(* PLC project Unnamed, Unknown Unnamed 1 *)
(* stored: creationDateTime 2025-11-06T09:56:44, modificationDateTime 2025-11-07T13:27:40 *)

TYPE TrafficLightStruct : STRUCT
  Safe : BOOL := True;
  LightRed : BOOL := False;
  LightGreen : BOOL := False;
  LightYellow : BOOL := False;
END_STRUCT;
END_TYPE

TYPE CrossWalkStruct : STRUCT
  Safe : BOOL := True;
  WalkLight : BOOL := False;
  DontWalkLight : BOOL := False;
END_STRUCT;
END_TYPE

TYPE InputMapStruct : STRUCT
  StartButton : BOOL := False;
  StopButton : BOOL := True;
  ResetButton : BOOL := False;
  CrossButton : BOOL := False;
  RedLightSensor : BOOL := True;
  GreenLightSensor : BOOL := True;
  YellowLightSensor : BOOL := True;
  WalkLightSensor : BOOL := True;
  DontWalkLightSensor : BOOL := True;
END_STRUCT;
END_TYPE

PROGRAM input_mapping0
  VAR_EXTERNAL
    DI_PB1 : BOOL;
    DI_PB2 : BOOL;
    DI_PB3 : BOOL;
    DI_PB4 : BOOL;
    DI_LightSensor1 : BOOL;
    DI_LightSensor2 : BOOL;
    DI_LightSensor3 : BOOL;
    DI_LightSensor4 : BOOL;
    DI_LightSensor5 : BOOL;
    InputMapGlobal : InputMapStruct;
  END_VAR

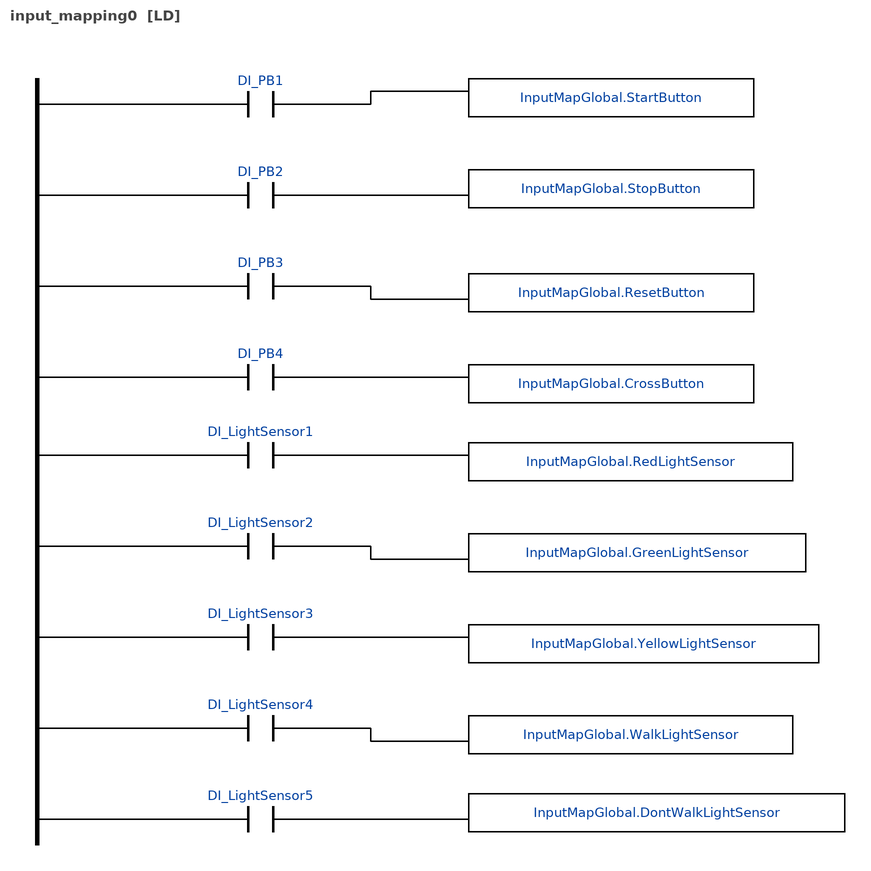
(* LD diagram, written out as Structured Text *)
InputMapGlobal.StartButton := DI_PB1;
InputMapGlobal.StopButton := DI_PB2;
InputMapGlobal.CrossButton := DI_PB4;
InputMapGlobal.RedLightSensor := DI_LightSensor1;
InputMapGlobal.GreenLightSensor := DI_LightSensor2;
InputMapGlobal.ResetButton := DI_PB3;
InputMapGlobal.YellowLightSensor := DI_LightSensor3;
InputMapGlobal.WalkLightSensor := DI_LightSensor4;
InputMapGlobal.DontWalkLightSensor := DI_LightSensor5;
END_PROGRAM

PROGRAM SystemControl
  VAR_EXTERNAL
    InputMapGlobal : InputMapStruct;
    Safe : BOOL;
  END_VAR
  VAR
    StartButton : BOOL;
    StopButton : BOOL;
  END_VAR
  VAR_EXTERNAL
    Running : BOOL;
  END_VAR

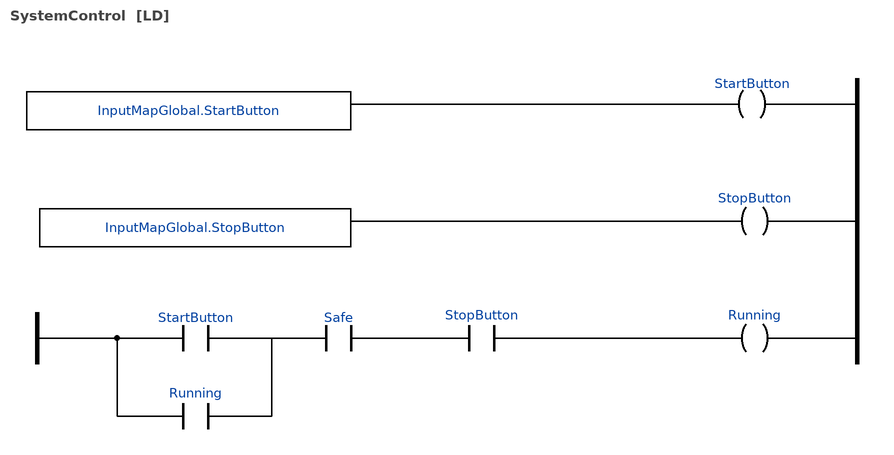
(* LD diagram, written out as Structured Text *)
StartButton := InputMapGlobal.StartButton;
StopButton := InputMapGlobal.StopButton;
Running := (StartButton OR Running) AND Safe AND StopButton;
END_PROGRAM

FUNCTION_BLOCK Flasher
  VAR_INPUT
    OnTime : TIME;
    OffTime : TIME;
  END_VAR
  VAR
    TON0 : TON;
    TOF0 : TOF;
  END_VAR
  VAR_OUTPUT
    F_On : BOOL;
  END_VAR

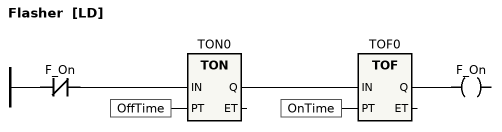
(* LD diagram, written out as Structured Text *)
TON0(IN := NOT F_On, PT := OffTime);
TOF0(IN := TON0.Q, PT := OnTime);
F_On := TOF0.Q;
END_FUNCTION_BLOCK

PROGRAM TrafficLightControl
  VAR_EXTERNAL
    Running : BOOL;
    Safe : BOOL;
    InputMapGlobal : InputMapStruct;
    TrafficLightState : TrafficLightStruct;
  END_VAR
  VAR
    LightCycle : BOOL := False;
    BlinkCycle : BOOL := False;
  END_VAR
  VAR
    Fault_RedLight AT %QX1.0 : BOOL := False;
    Fault_GreenLight AT %QX1.1 : BOOL := False;
    Fault_YellowLight AT %QX1.2 : BOOL := False;
  END_VAR
  VAR
    RedLight : BOOL := False;
    GreenLight : BOOL := False;
    YellowLight : BOOL := False;
    Reset : BOOL := False;
    ResetButton : BOOL := False;
    RedLightSensor : BOOL := False;
    GreenLightSensor : BOOL := False;
    YellowLightSensor : BOOL := False;
    T_YellowLight : TON;
    T_RedLight : TON;
    T_GreenLight : TON;
    Flasher1 : Flasher;
  END_VAR
  VAR  (* added by the conversion: wires and edge detectors of the diagram *)
    R_TRIG1 : R_TRIG;
  END_VAR

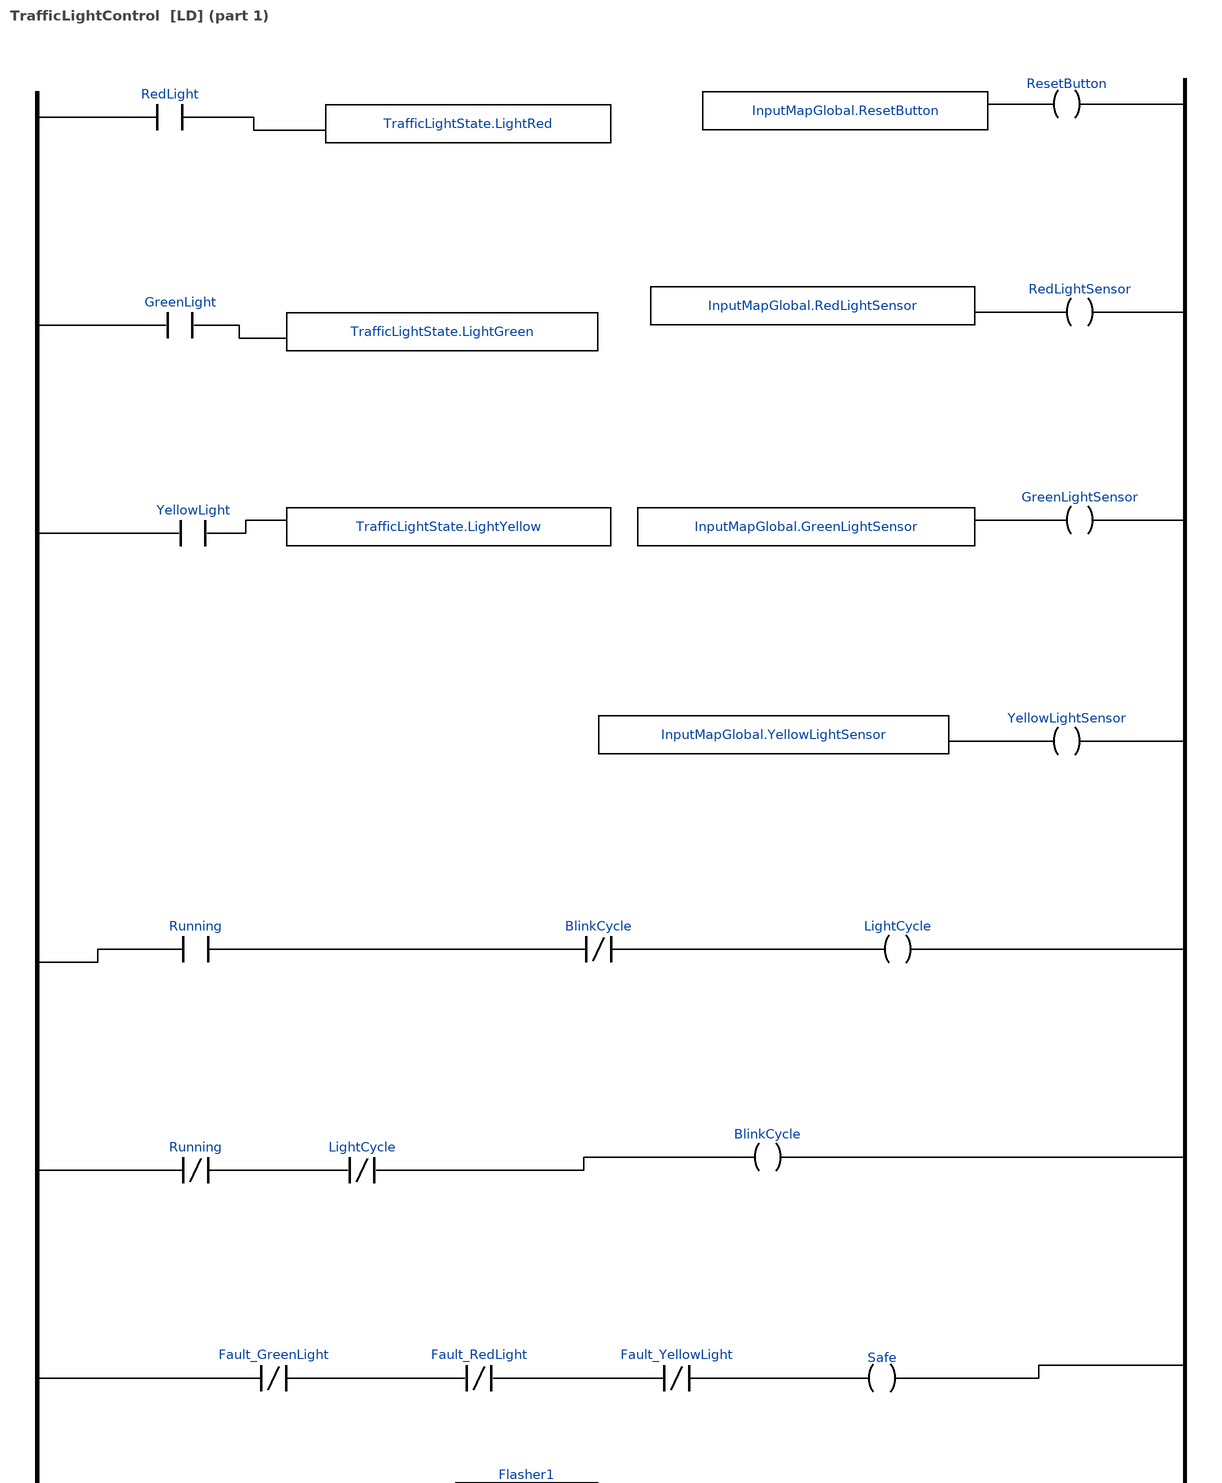
(* LD diagram, written out as Structured Text *)
ResetButton := InputMapGlobal.ResetButton;
RedLightSensor := InputMapGlobal.RedLightSensor;
GreenLightSensor := InputMapGlobal.GreenLightSensor;
YellowLightSensor := InputMapGlobal.YellowLightSensor;
LightCycle := Running AND NOT BlinkCycle;
BlinkCycle := NOT Running AND NOT LightCycle;
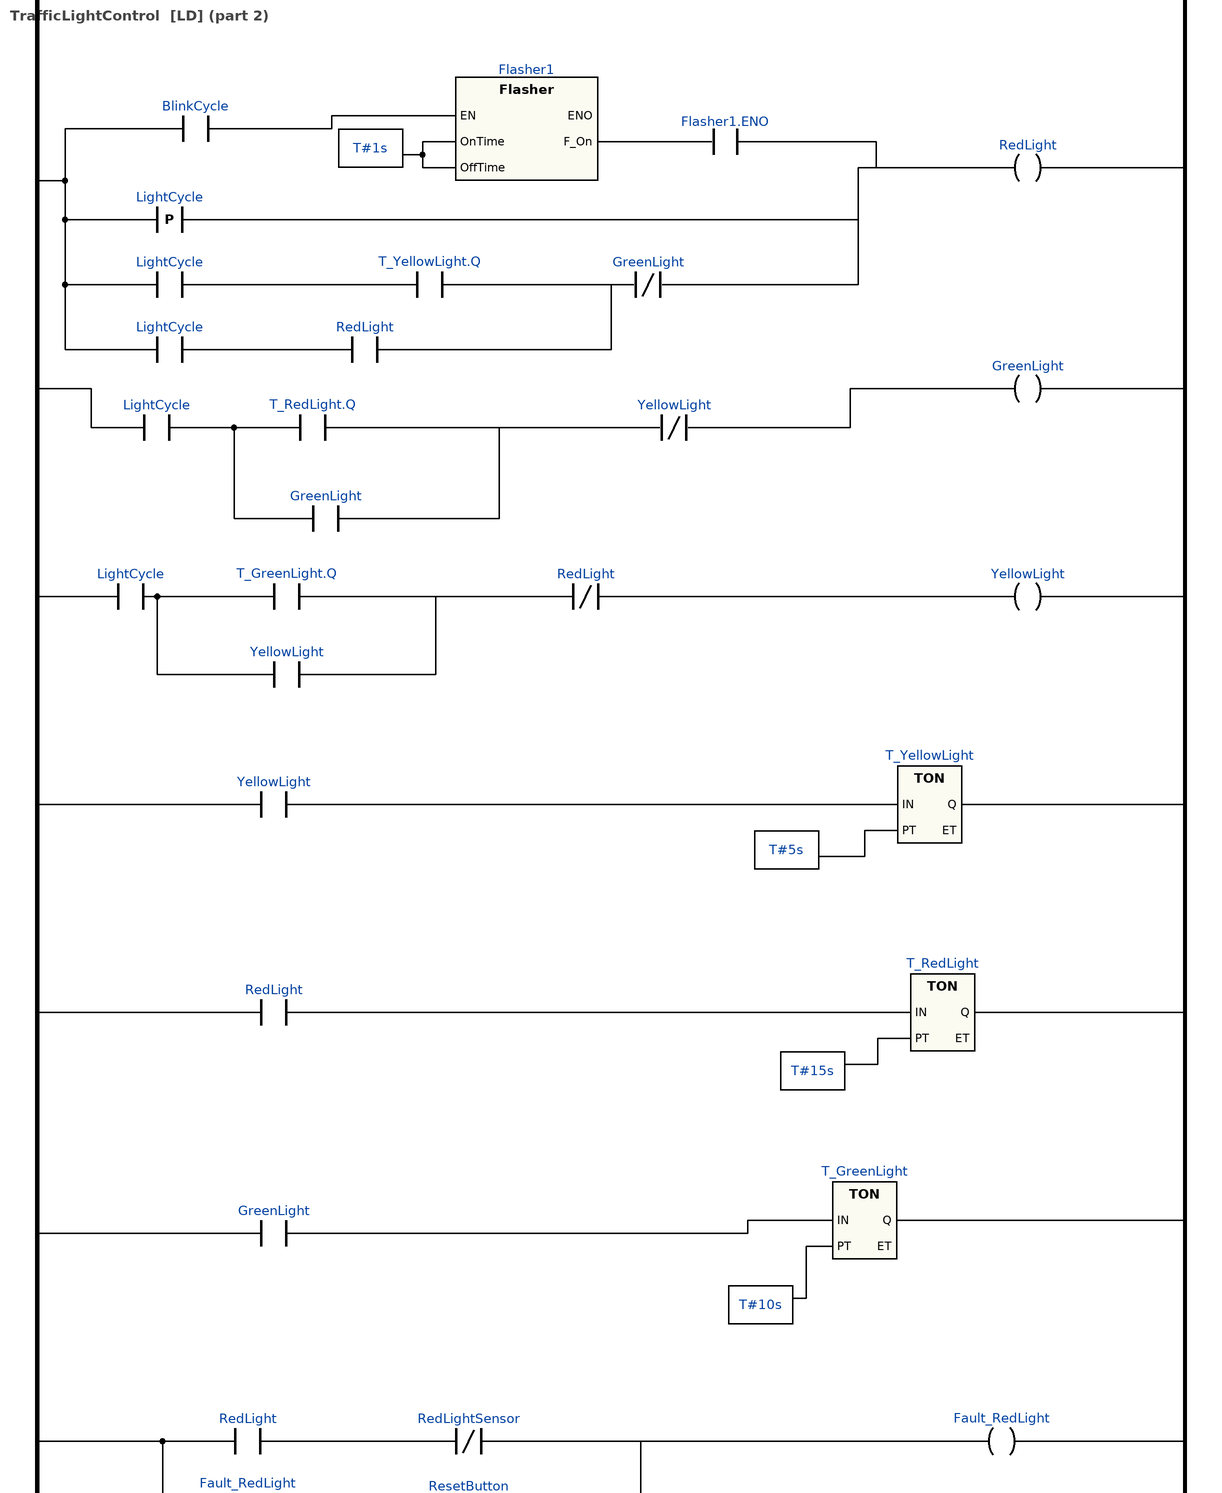
GreenLight := LightCycle AND (T_RedLight.Q OR GreenLight) AND NOT YellowLight;
YellowLight := LightCycle AND (T_GreenLight.Q OR YellowLight) AND NOT RedLight;
R_TRIG1(CLK := LightCycle);
Flasher1(EN := BlinkCycle, OnTime := T#1s, OffTime := T#1s);
RedLight := R_TRIG1.Q OR LightCycle AND (T_YellowLight.Q OR RedLight) AND NOT GreenLight OR Flasher1.F_On AND Flasher1.ENO;
Fault_RedLight := RedLight AND NOT RedLightSensor OR Fault_RedLight AND NOT ResetButton;
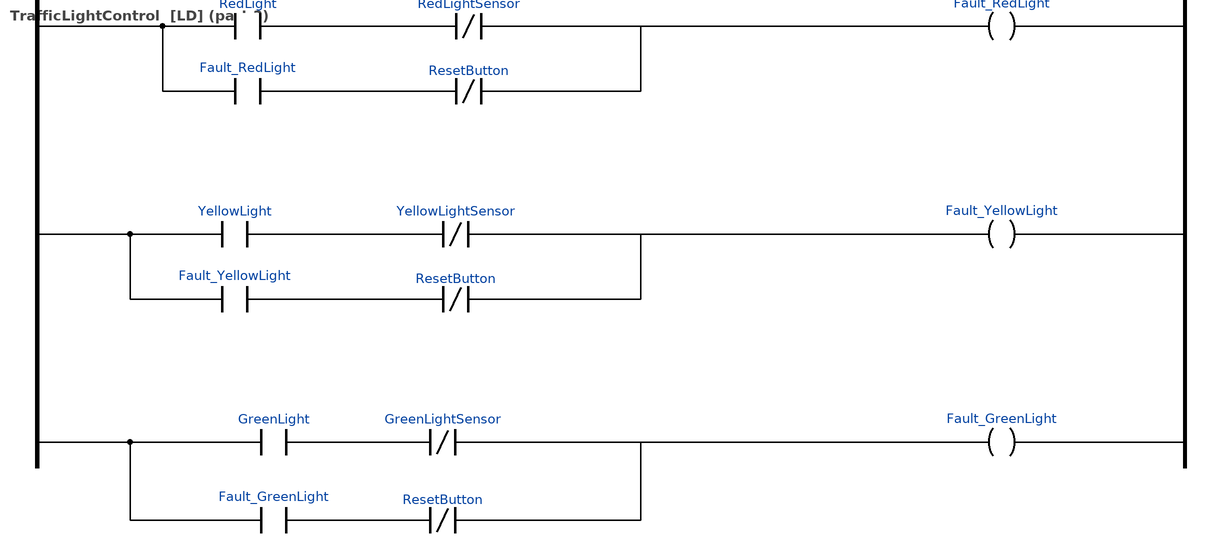
Fault_YellowLight := YellowLight AND NOT YellowLightSensor OR Fault_YellowLight AND NOT ResetButton;
Fault_GreenLight := GreenLight AND NOT GreenLightSensor OR Fault_GreenLight AND NOT ResetButton;
Safe := NOT Fault_GreenLight AND NOT Fault_RedLight AND NOT Fault_YellowLight;
TrafficLightState.LightRed := RedLight;
TrafficLightState.LightGreen := GreenLight;
TrafficLightState.LightYellow := YellowLight;
T_YellowLight(IN := YellowLight, PT := T#5s);
T_RedLight(IN := RedLight, PT := T#15s);
T_GreenLight(IN := GreenLight, PT := T#10s);
END_PROGRAM

PROGRAM CrosswalkControl
  VAR_EXTERNAL
    InputMapGlobal : InputMapStruct;
    CrossWalkState : CrossWalkStruct;
    TrafficLightState : TrafficLightStruct;
    Running : BOOL;
    Safe : BOOL;
  END_VAR
  VAR
    CrosswalkButton : BOOL := False;
    ResetButton : BOOL := False;
    WalkLight : BOOL := False;
    DontWalkLight : BOOL := False;
    CrosswalkSequence : BOOL := False;
    CrosswalkSequence_End : BOOL := False;
    WalkLightFault : BOOL := False;
    DontWalkLightFault : BOOL := False;
    WaitForWalk : BOOL := False;
    Walk : BOOL := False;
    StopWalk : BOOL := False;
    RedLight : BOOL := False;
    GreenLight : BOOL := False;
    T_Walk : TON;
    Flasher0 : Flasher;
    DontWalkLightSensor : BOOL;
    WalkLightSensor : BOOL;
  END_VAR
  VAR  (* added by the conversion: wires and edge detectors of the diagram *)
    R_TRIG1 : R_TRIG;
    R_TRIG2 : R_TRIG;
    R_TRIG3 : R_TRIG;
  END_VAR

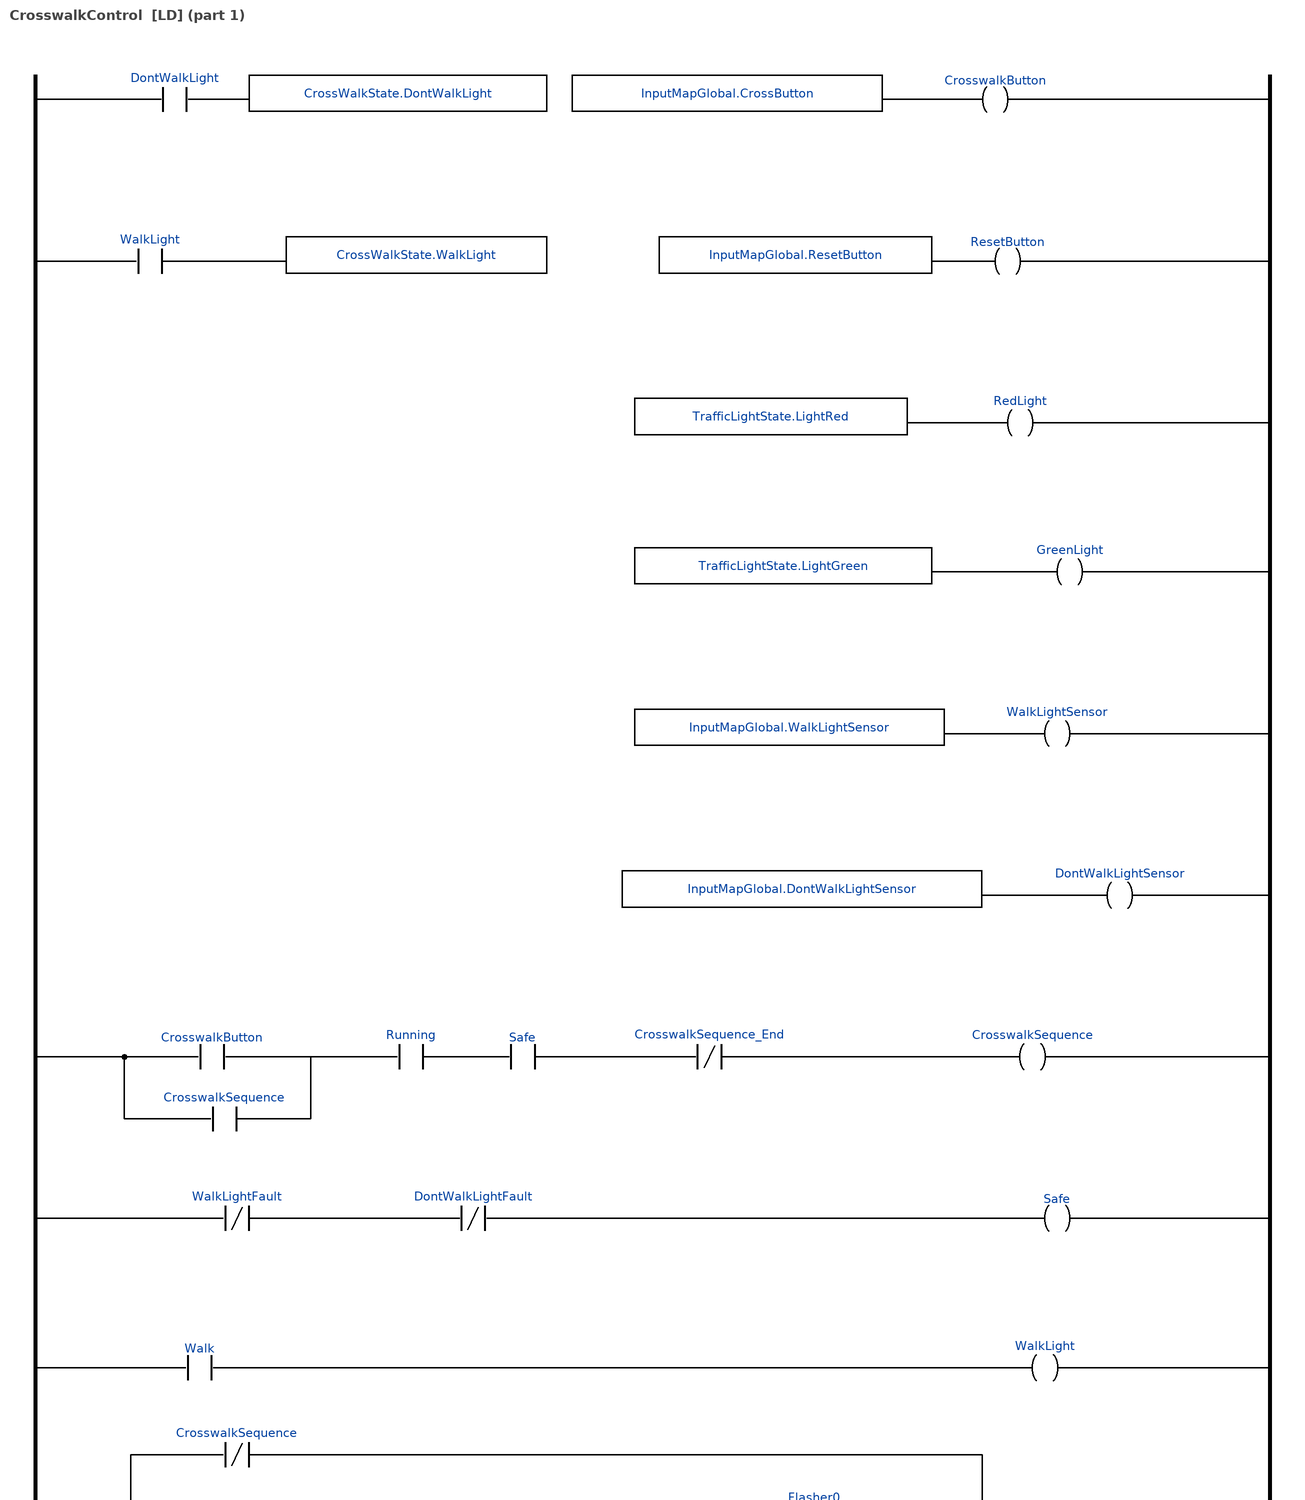
(* LD diagram, written out as Structured Text *)
CrosswalkButton := InputMapGlobal.CrossButton;
ResetButton := InputMapGlobal.ResetButton;
CrossWalkState.DontWalkLight := DontWalkLight;
CrossWalkState.WalkLight := WalkLight;
CrosswalkSequence := (CrosswalkButton OR CrosswalkSequence) AND Running AND Safe AND NOT CrosswalkSequence_End;
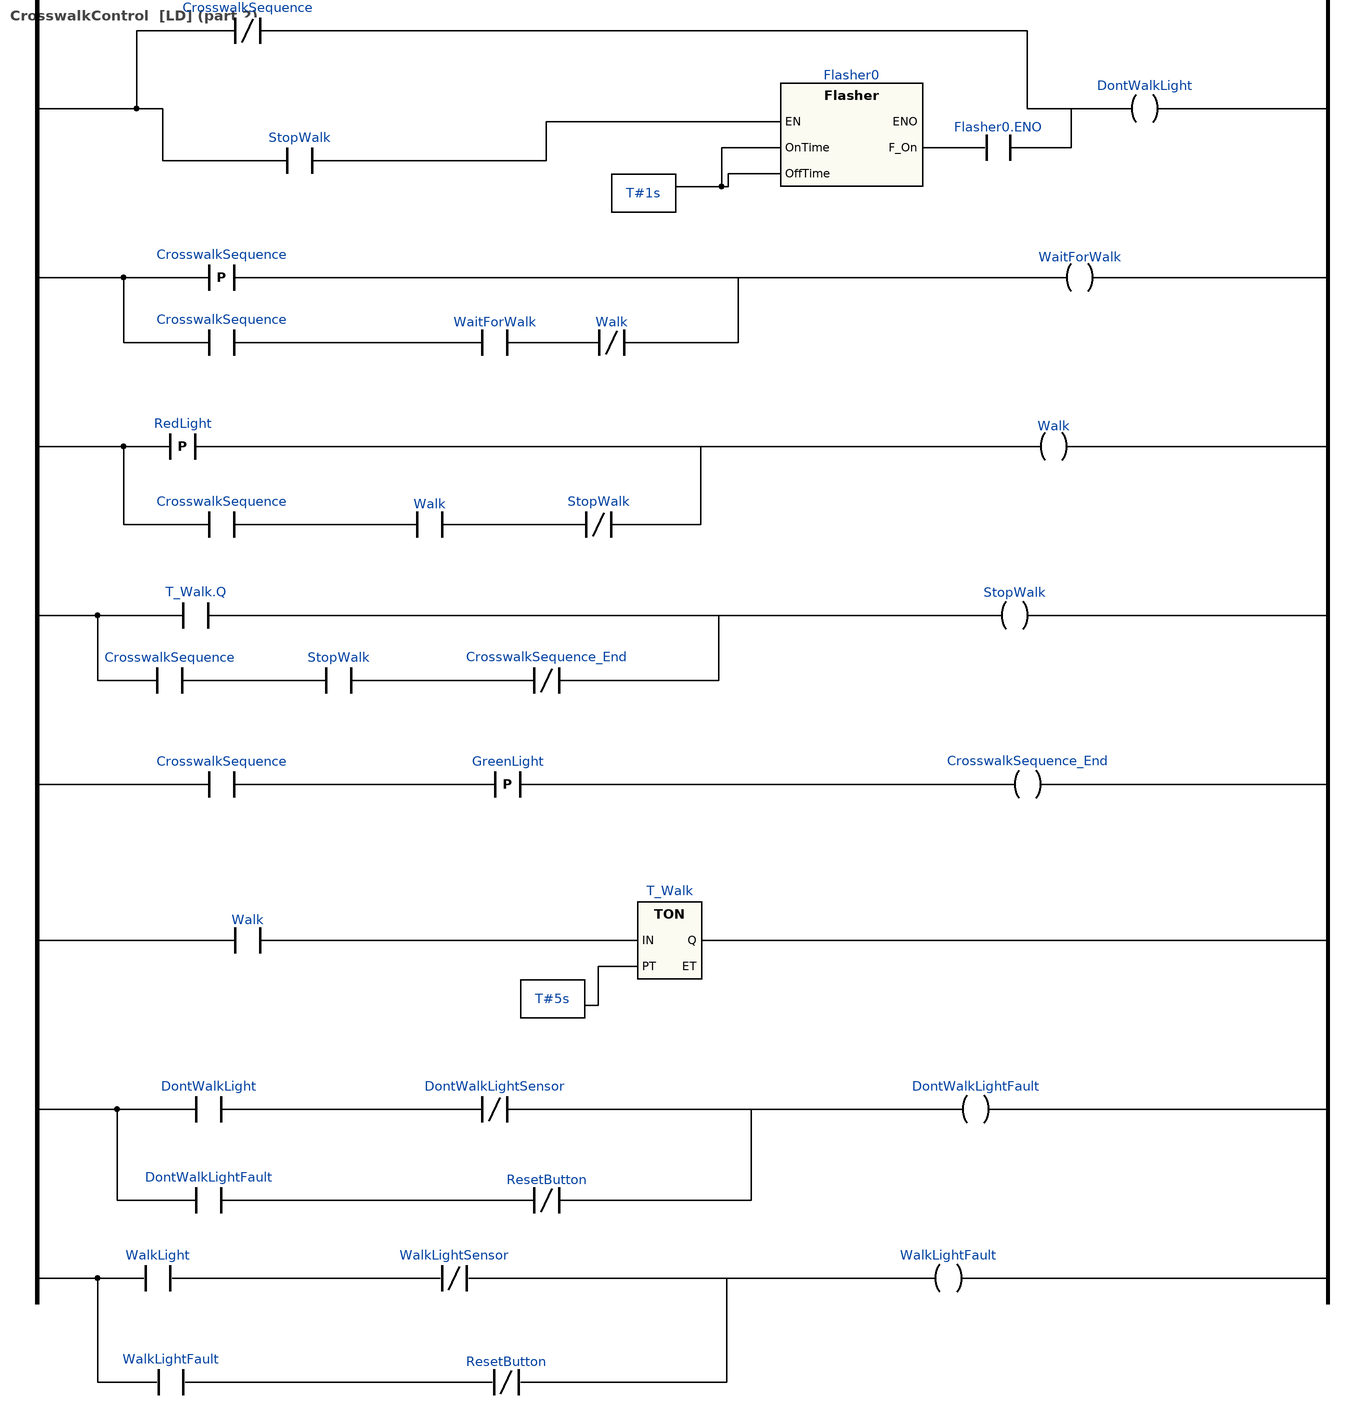
R_TRIG1(CLK := CrosswalkSequence);
WaitForWalk := R_TRIG1.Q OR CrosswalkSequence AND WaitForWalk AND NOT Walk;
RedLight := TrafficLightState.LightRed;
R_TRIG2(CLK := RedLight);
Walk := CrosswalkSequence AND Walk AND NOT StopWalk OR R_TRIG2.Q;
StopWalk := T_Walk.Q OR CrosswalkSequence AND StopWalk AND NOT CrosswalkSequence_End;
GreenLight := TrafficLightState.LightGreen;
R_TRIG3(CLK := GreenLight);
CrosswalkSequence_End := CrosswalkSequence AND R_TRIG3.Q;
Safe := NOT WalkLightFault AND NOT DontWalkLightFault;
WalkLight := Walk;
Flasher0(EN := StopWalk, OnTime := T#1s, OffTime := T#1s);
DontWalkLight := NOT CrosswalkSequence OR Flasher0.F_On AND Flasher0.ENO;
WalkLightSensor := InputMapGlobal.WalkLightSensor;
DontWalkLightSensor := InputMapGlobal.DontWalkLightSensor;
DontWalkLightFault := DontWalkLight AND NOT DontWalkLightSensor OR DontWalkLightFault AND NOT ResetButton;
WalkLightFault := WalkLight AND NOT WalkLightSensor OR WalkLightFault AND NOT ResetButton;
T_Walk(IN := Walk, PT := T#5s);
END_PROGRAM

PROGRAM output_mapping
  VAR_EXTERNAL
    TrafficLightState : TrafficLightStruct;
    CrosswalkState : CrossWalkStruct;
    DQ_LightRed : BOOL;
    DQ_LightGreen : BOOL;
    DQ_LightYellow : BOOL;
    DQ_LightWalk : BOOL;
    DQ_LightDontWalk : BOOL;
  END_VAR

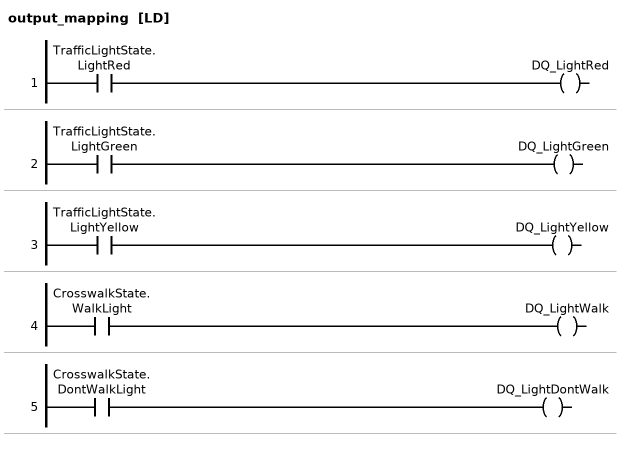
(* LD diagram, written out as Structured Text *)
DQ_LightRed := TrafficLightState.LightRed;
DQ_LightGreen := TrafficLightState.LightGreen;
DQ_LightYellow := TrafficLightState.LightYellow;
DQ_LightWalk := CrosswalkState.WalkLight;
DQ_LightDontWalk := CrosswalkState.DontWalkLight;
END_PROGRAM

CONFIGURATION Config0
  VAR_GLOBAL
    DI_PB1 AT %IX0.0 : BOOL := False;
    DI_PB2 AT %IX0.1 : BOOL := True;  (* Wired NC *)
    DI_PB3 AT %IX0.2 : BOOL := False;
    DI_PB4 AT %IX0.3 : BOOL := False;
    DI_LightSensor1 AT %IX0.4 : BOOL := True;
    DI_LightSensor2 AT %IX0.5 : BOOL := True;
    DI_LightSensor3 AT %IX0.6 : BOOL := True;
    DI_LightSensor4 AT %IX0.7 : BOOL := True;
    DI_LightSensor5 AT %IX1.0 : BOOL := True;
    DQ_LightRed AT %QX0.0 : BOOL := False;
    DQ_LightGreen AT %QX0.1 : BOOL := False;
    DQ_LightYellow AT %QX0.2 : BOOL := False;
    DQ_LightWalk AT %QX0.3 : BOOL := False;
    DQ_LightDontWalk AT %QX0.4 : BOOL := False;
    Running AT %QX0.5 : BOOL := False;  (* Shows system is running. Has HMI output *)
    Safe AT %QX0.6 : BOOL := True;  (* Shows system is safe. Has HMI output *)
    TrafficLightState : TrafficLightStruct;
    CrossWalkState : CrossWalkStruct;
    InputMapGlobal : InputMapStruct;
  END_VAR
  RESOURCE Res0 ON PLC
    TASK task0(INTERVAL := T#20ms, PRIORITY := 0);
    PROGRAM input_map WITH task0 : input_mapping0;
    PROGRAM system_control WITH task0 : SystemControl;
    PROGRAM trafficlight_control WITH task0 : TrafficLightControl;
    PROGRAM crosswalk_control WITH task0 : CrosswalkControl;
    PROGRAM output_map WITH task0 : output_mapping;
  END_RESOURCE
END_CONFIGURATION
